TYPE (* A +-11-bit Subrange Data Type *)
  (* Standard: 61131-3 *)
  (* Version 0.0, 2004-01-02, JHC, Rockwell Automation, Derived from Subrange template. *)
  (* Compiler header: package fb.rt.test; *)
  (* Compiler Java IBM VisualAge 3.0 *)
  (* ASN.1 tag PRIVATE 10 *)
  SUBR12 : INT(-4095..4095);
END_TYPE
